// TIA Portal V20 export
// export: Created 2025-12-01T14:56:17.4883297Z, ExportSetting None, DisplayName Totally Integrated Automation Portal, DisplayVersion V20 Update 3, DisplayName TIA Portal Openness, DisplayVersion V20 Update 3, DisplayName TIA Portal Version Control Interface, DisplayVersion V20 Update 3, DisplayName STEP 7 Professional, DisplayVersion V20 Update 3, DisplayName STEP 7 Safety, DisplayVersion V20 Update 2, DisplayName WinCC Basic/Comfort/Advanced, DisplayVersion V20 Update 3, DisplayName WinCC Professional, DisplayVersion V20 Update 3, DisplayName WinCC Unified, DisplayVersion V20 Update 3
TYPE "Interlock_Paletas_PLC_IKPAL"
   STRUCT
      BitDeVida : Bool;
      Libre_01 : Bool;
      Libre_02 : Bool;
      Libre_03 : Bool;
      Libre_04 : Bool;
      Libre_05 : Bool;
      Libre_06 : Bool;
      Libre_07 : Bool;
      Salida_Automatico : Bool;
      Salida_Marcha : Bool;
      Salida_Error : Bool;
      PaletaVacia_Automatico : Bool;
      PaletaVacia_Marcha : Bool;
      PaletaVacia_Error : Bool;
      Preformado_Automatico : Bool;
      Preformado_Marcha : Bool;
      Preformado_Error : Bool;
      Libre_21 : Bool;
      Libre_22 : Bool;
      Libre_23 : Bool;
      Libre_24 : Bool;
      Libre_25 : Bool;
      Libre_26 : Bool;
      Libre_27 : Bool;
      Libre_30 : Bool;
      Libre_31 : Bool;
      Libre_32 : Bool;
      Libre_33 : Bool;
      Libre_34 : Bool;
      Libre_35 : Bool;
      Libre_36 : Bool;
      Libre_37 : Bool;
      Reserva_Array_04_B04 : Array[1..4] of Byte;
      PermisoPaleta_NXT : Bool;
      FinPaleta_NTXT : Bool;
      PermisoPaleta_NXT_Manual_Av : Bool;
      PermisoPaleta_NXT_Manual_Ret : Bool;
      Libre_84 : Bool;
      Libre_85 : Bool;
      Libre_86 : Bool;
      Libre_87 : Bool;
      PermisoExtenderHorquillas : Bool;
      PermisoCentrarHorquillas : Bool;
      PermisoAperturaPuertas : Bool;
      MaquetaArriba : Bool;
      MaquetaAbajo : Bool;
      Libre_95 : Bool;
      Libre_96 : Bool;
      Libre_97 : Bool;
      AvisoPreformado_PRV : Bool;
      OrdenMarchaPreformado_PRV : Bool;
      AvisoPreformado_PRV_Manual_Av : Bool;
      AvisoPreformado_PRV_Manual_Ret : Bool;
      Libre_104 : Bool;
      Libre_105 : Bool;
      Libre_106 : Bool;
      Libre_107 : Bool;
      Libre_110 : Bool;
      Libre_111 : Bool;
      Libre_112 : Bool;
      Libre_113 : Bool;
      Libre_114 : Bool;
      Libre_115 : Bool;
      Libre_116 : Bool;
      Libre_117 : Bool;
      CotaAlturaPreformado : UInt;
      Reserva_Array_04_B14 : Array[1..4] of Byte;
      MatriculaPreformado : Array[1..10] of Byte;
      MckeyPreformado : Array[1..8] of Byte;
      Reserva_Array_02_B36 : Array[1..2] of Byte;
      MatriculaPaletaVacia : Array[1..10] of Byte;
      MckeyPaletaVacia : Array[1..8] of Byte;
   END_STRUCT;
END_TYPE
